{attribute addProperty BoxType "EL2535-0103-0023"}
{attribute addProperty Id "PWM_Status_ChannelAT %I*ARRAY[0..1] OF PWM_Status_Channel_1DED96923240PWM_Control_ChannelAT %Q*ARRAY[0..2] OF PWM_Control_Channel_253BEA616480WcStateAT %I*WcState_98A4DF7520.250InfoDataAT %I*InfoData_BC63D37F80100"}
{attribute addProperty CRC "1312458753"}
{attribute addProperty SizeInBites "178"}
{attribute addProperty SizeInBytes "22.25"}
TYPE EL2535_93E74954 :
STRUCT
	{attribute addProperty Name "PWM_Status_Channel"}
	PWM_Status_Channel : ARRAY[0..1] OF PWM_Status_Channel_1DED9692;
	{attribute addProperty Name "PWM_Control_Channel"}
	PWM_Control_Channel : ARRAY[0..2] OF PWM_Control_Channel_253BEA61;
	{attribute addProperty Name "WcState"}
	WcState : WcState_98A4DF75;
	{attribute addProperty Name "InfoData"}
	InfoData : InfoData_BC63D37F;
END_STRUCT
END_TYPE

(* stored: Version 1.2.0.0, ProductVersion 3.1.4024.9
   DUT EL2535_93E74954: Id {416eb54c-4de4-4818-8fe4-35046588dd41} *)
